(* Logix 5000 project; controller Safety vendor 1 type 14 code 86 rev 19.11; software revision 19.01; part 8 of 17 *)
(* tags used below, declared in another part *)
   ESTOP_x201PB040 : DCI_STOP;   // OS1 Line EStop Pushbutton
   ESTOP_x201PB040_Flt : ALIAS FOR Flt_Estops.0;   // OS1 Line EStop Pushbutton Fault ( 1= Fault)
   ESTOP_x211PB040 : DCI_STOP;   // OS2 Line EStop Pushbutton
   ESTOP_x211PB040_Flt : ALIAS FOR Flt_Estops.1;   // OS2 Line EStop Pushbutton Fault ( 1= Fault)
   ESTOP_x221PB040 : DCI_STOP;   // OS3 Line EStop Pushbutton
   ESTOP_x221PB040_Flt : ALIAS FOR Flt_Estops.2;   // OS3 Line EStop Pushbutton Fault ( 1= Fault)
   ESTOP_x231PB040 : DCI_STOP;   // OS4N Line EStop Pushbutton
   ESTOP_x231PB040_Flt : ALIAS FOR Flt_Estops.3;   // OS4N Line EStop Pushbutton Fault ( 1= Fault)
   ESTOP_x241PB040 : DCI_STOP;   // OS4S Line EStop Pushbutton
   ESTOP_x241PB040_Flt : ALIAS FOR Flt_Estops.4;   // OS4S Line EStop Pushbutton Fault ( 1= Fault)
   ESTOP_x251PB040 : DCI_STOP;   // OS5 Line EStop Pushbutton
   ESTOP_x251PB040_Flt : ALIAS FOR Flt_Estops.5;   // OS5 Line EStop Pushbutton Fault ( 1= Fault)
   ESTOP_x261PB040 : DCI_STOP;   // OS6 Line EStop Pushbutton
   ESTOP_x261PB040_Flt : ALIAS FOR Flt_Estops.6;   // OS6 Line EStop Pushbutton Fault ( 1= Fault)
   ESTOP_x271PB040 : DCI_STOP;   // OS8 Line EStop Pushbutton
   ESTOP_x271PB040_Flt : ALIAS FOR Flt_Estops.7;   // OS8 Line EStop Pushbutton Fault ( 1= Fault)
   ESTOP_x281PB040 : DCI_STOP;   // OS9 Line EStop Pushbutton
   ESTOP_x301PB040 : DCI_STOP;   // OS13 Line EStop Pushbutton
   ESTOP_x311PB040 : DCI_STOP;   // OS14 Line EStop Pushbutton
   ESTOP_x311PB130 : DCI_STOP;   // OS14 Shear Estop Pushbutton
   ESTOP_x321PB040 : DCI_STOP;   // OS15 Line EStop Pushbutton
   ESTOP_x331PB040 : DCI_STOP;   // OS16 Line EStop Pushbutton
   ESTOP_x480PB550 : DCI_STOP;   // DPD (In Pit) Line EStop Pushbutton
   ESTOP_x519LS470 : DCI_STOP;   // G1 Tripwire Line EStop
   ESTOP_x533PB470 : DCI_STOP;   // H1 Line EStop Pushbutton
   Line_TotalMode : BOOL;   // Line TOTAL Mode ( 1= Total Mode) (0 = Coil to Coil)
   LineSts : UDT_SysStatus;
   OS1_EstopRstCmd : BOOL;   // OS1 Estop Reset Command ( 1= Reset Cmd)
   OS1_FltRstCmd : BOOL;   // OS1 Fault Reset Command ( 1= Reset Cmd)
   OS1_No_EStops : BOOL;   // OS1 No Estops ( 1= OK)
   OS2_EstopRstCmd : BOOL;   // OS2 Estop Reset Command ( 1= Reset Cmd)
   OS2_FltRstCmd : BOOL;   // OS2 Fault Reset Command ( 1= Reset Cmd)
   OS2_No_EStops : BOOL;   // OS2 No Estops ( 1= OK)
   OS3_EstopRstCmd : BOOL;   // OS3 Estop Reset Command ( 1= Reset Cmd)
   OS3_FltRstCmd : BOOL;   // OS3 Fault Reset Command ( 1= Reset Cmd)
   OS3_No_EStops : BOOL;   // OS3 No Estops ( 1= OK)
   OS4_EstopRstCmd : BOOL;   // OS4 Estop Reset Command ( 1= Reset Cmd)
   OS4_FltRstCmd : BOOL;   // OS4 Fault Reset Command ( 1= Reset Cmd)
   OS4_No_EStops : BOOL;   // OS4 No Estops ( 1= OK)
   OS5_EstopRstCmd : BOOL;   // OS5 Estop Reset Command ( 1= Reset Cmd)
   OS5_FltRstCmd : BOOL;   // OS5 Fault Reset Command ( 1= Reset Cmd)
   OS5_No_EStops : BOOL;   // OS5 No Estops ( 1= OK)
   OS6_EstopRstCmd : BOOL;   // OS6 Estop Reset Command ( 1= Reset Cmd)
   OS6_FltRstCmd : BOOL;   // OS6 Fault Reset Command ( 1= Reset Cmd)
   OS6_No_EStops : BOOL;   // OS6 No Estops ( 1= OK)
   OS8_EstopRstCmd : BOOL;   // OS8 Estop Reset Command ( 1= Reset Cmd)
   OS8_FltRstCmd : BOOL;   // OS8 Fault Reset Command ( 1= Reset Cmd)
   OS8_No_EStops : BOOL;   // OS8 No Estops ( 1= OK)
   x201PB040a : ALIAS FOR OS1:1:I.Pt00Data;   // Line Emergency Stop PB
   x201PB040b : ALIAS FOR OS1:1:I.Pt01Data;   // Line Emergency Stop PB
   x211PB040a : ALIAS FOR OS2:1:I.Pt00Data;   // Line Emergency Stop PB
   x211PB040b : ALIAS FOR OS2:1:I.Pt01Data;   // Line Emergency Stop PB
   x221PB040a : ALIAS FOR OS3:1:I.Pt00Data;   // Emergency Stop PB
   x221PB040b : ALIAS FOR OS3:1:I.Pt01Data;   // Emergency Stop PB
   x231PB040a : ALIAS FOR OS4N:1:I.Pt00Data;   // Emergency Stop PB
   x231PB040b : ALIAS FOR OS4N:1:I.Pt01Data;   // Emergency Stop PB
   x241PB040a : ALIAS FOR OS4S:1:I.Pt00Data;   // Emergency Stop PBMc_A_Run1_A
   x241PB040b : ALIAS FOR OS4S:1:I.Pt01Data;   // Emergency Stop PBMc_A_Run1_A
   x251PB040a : ALIAS FOR OS5:1:I.Pt00Data;   // Emergency Stop PB
   x251PB040b : ALIAS FOR OS5:1:I.Pt01Data;   // Emergency Stop PB
   x261PB040a : ALIAS FOR OS6:1:I.Pt00Data;   // Emergency Stop PB
   x261PB040b : ALIAS FOR OS6:1:I.Pt01Data;   // Emergency Stop PB
   x271PB040a : ALIAS FOR OS8:1:I.Pt00Data;   // Emergency Stop PB
   x271PB040b : ALIAS FOR OS8:1:I.Pt01Data;   // Emergency Stop PB

PROGRAM Estops   (* main routine A00_Main *)
// Estop PB's

ROUTINE A00_Main   (* ladder *)
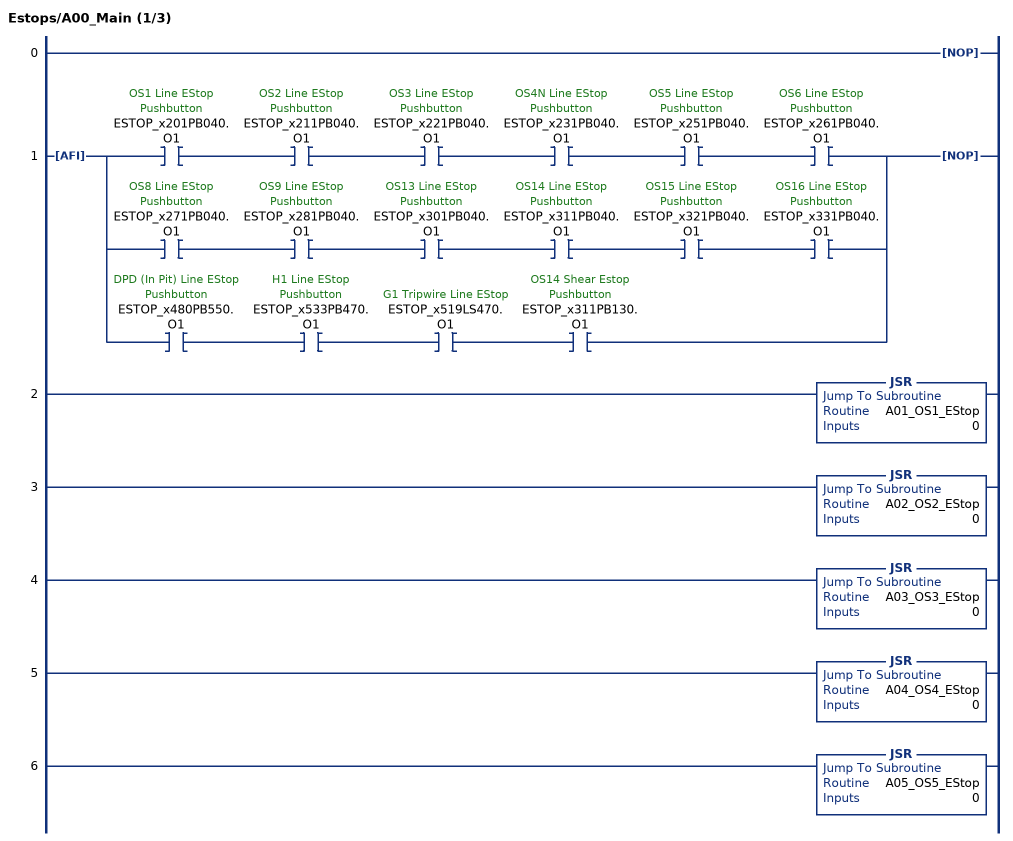
   0: NOP();
   1: AFI()[XIC(ESTOP_x201PB040.O1) XIC(ESTOP_x211PB040.O1) XIC(ESTOP_x221PB040.O1) XIC(ESTOP_x231PB040.O1) XIC(ESTOP_x251PB040.O1) XIC(ESTOP_x261PB040.O1) ,XIC(ESTOP_x271PB040.O1) XIC(ESTOP_x281PB040.O1) XIC(ESTOP_x301PB040.O1) XIC(ESTOP_x311PB040.O1) XIC(ESTOP_x321PB040.O1) XIC(ESTOP_x331PB040.O1) ,XIC(ESTOP_x480PB550.O1) XIC(ESTOP_x533PB470.O1) XIC(ESTOP_x519LS470.O1) XIC(ESTOP_x311PB130.O1) ]NOP();
   2: JSR(A01_OS1_EStop,0);
   3: JSR(A02_OS2_EStop,0);
   4: JSR(A03_OS3_EStop,0);
   5: JSR(A04_OS4_EStop,0);
   6: JSR(A05_OS5_EStop,0);
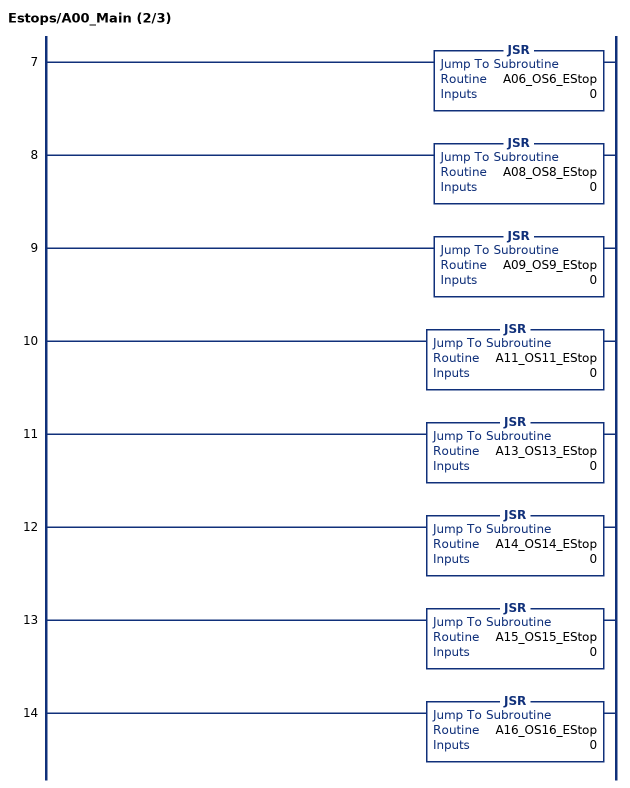
   7: JSR(A06_OS6_EStop,0);
   8: JSR(A08_OS8_EStop,0);
   9: JSR(A09_OS9_EStop,0);
   10: JSR(A11_OS11_EStop,0);
   11: JSR(A13_OS13_EStop,0);
   12: JSR(A14_OS14_EStop,0);
   13: JSR(A15_OS15_EStop,0);
   14: JSR(A16_OS16_EStop,0);
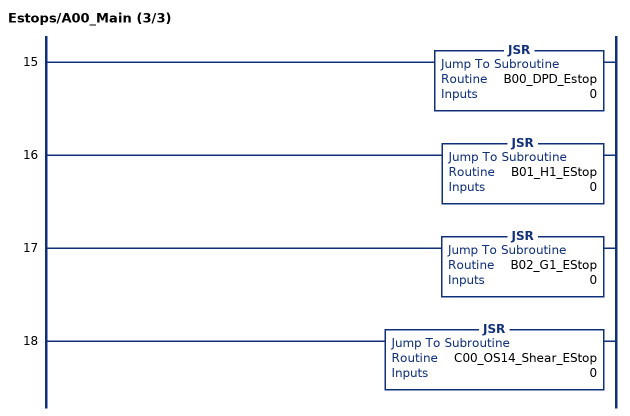
   15: JSR(B00_DPD_Estop,0);
   16: JSR(B01_H1_EStop,0);
   17: JSR(B02_G1_EStop,0);
   18: JSR(C00_OS14_Shear_EStop,0);
END_ROUTINE

ROUTINE A01_OS1_EStop   (* ladder *)
// OS1 Estops
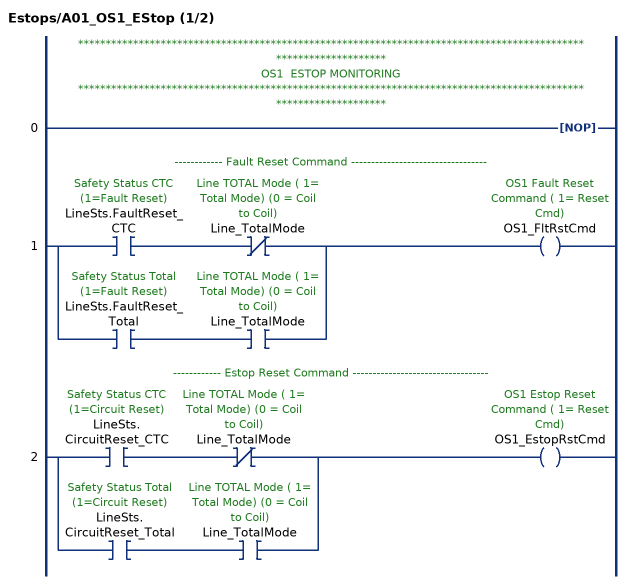
   // ****************************************************************************************************************
   // OS1  ESTOP MONITORING
   // ****************************************************************************************************************
   0: NOP();
   // ------------ Fault Reset Command ----------------------------------
   1: [XIC(LineSts.FaultReset_CTC) XIO(Line_TotalMode) ,XIC(LineSts.FaultReset_Total) XIC(Line_TotalMode) ]OTE(OS1_FltRstCmd);
   // ------------ Estop Reset Command ----------------------------------
   2: [XIC(LineSts.CircuitReset_CTC) XIO(Line_TotalMode) ,XIC(LineSts.CircuitReset_Total) XIC(Line_TotalMode) ]OTE(OS1_EstopRstCmd);
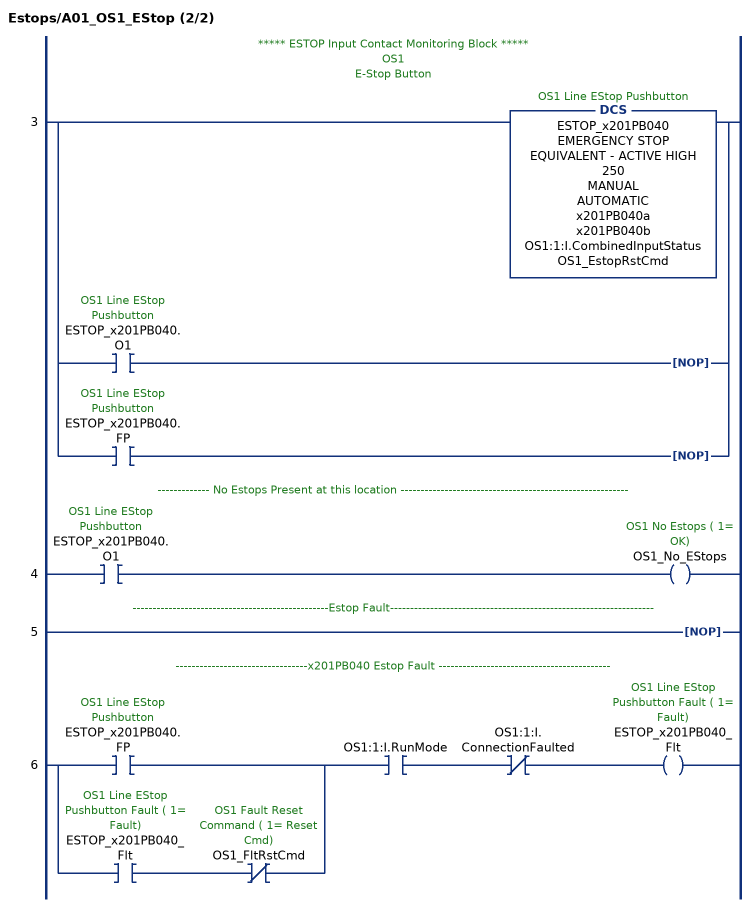
   // ***** ESTOP Input Contact Monitoring Block *****
   // OS1
   // E-Stop Button
   3: [DCS(ESTOP_x201PB040,EMERGENCY STOP,EQUIVALENT - ACTIVE HIGH,250,MANUAL,AUTOMATIC,x201PB040a,x201PB040b,OS1:1:I.CombinedInputStatus,OS1_EstopRstCmd) ,XIC(ESTOP_x201PB040.O1) NOP() ,XIC(ESTOP_x201PB040.FP) NOP() ];
   // ------------- No Estops Present at this location ---------------------------------------------------------
   4: XIC(ESTOP_x201PB040.O1)OTE(OS1_No_EStops);
   // -------------------------------------------------Estop Fault------------------------------------------------------------------
   5: NOP();
   // ---------------------------------x201PB040 Estop Fault -------------------------------------------
   6: [XIC(ESTOP_x201PB040.FP) ,XIC(ESTOP_x201PB040_Flt) XIO(OS1_FltRstCmd) ]XIC(OS1:1:I.RunMode)XIO(OS1:1:I.ConnectionFaulted)OTE(ESTOP_x201PB040_Flt);
END_ROUTINE

ROUTINE A02_OS2_EStop   (* ladder *)
// OS2 Estops
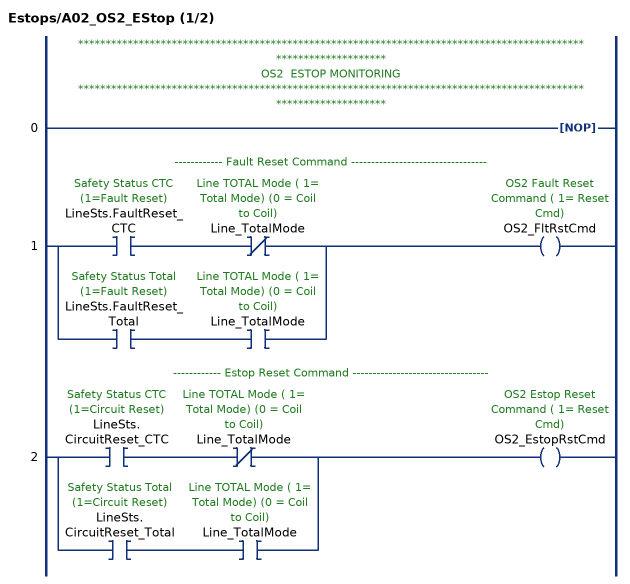
   // ****************************************************************************************************************
   // OS2  ESTOP MONITORING
   // ****************************************************************************************************************
   0: NOP();
   // ------------ Fault Reset Command ----------------------------------
   1: [XIC(LineSts.FaultReset_CTC) XIO(Line_TotalMode) ,XIC(LineSts.FaultReset_Total) XIC(Line_TotalMode) ]OTE(OS2_FltRstCmd);
   // ------------ Estop Reset Command ----------------------------------
   2: [XIC(LineSts.CircuitReset_CTC) XIO(Line_TotalMode) ,XIC(LineSts.CircuitReset_Total) XIC(Line_TotalMode) ]OTE(OS2_EstopRstCmd);
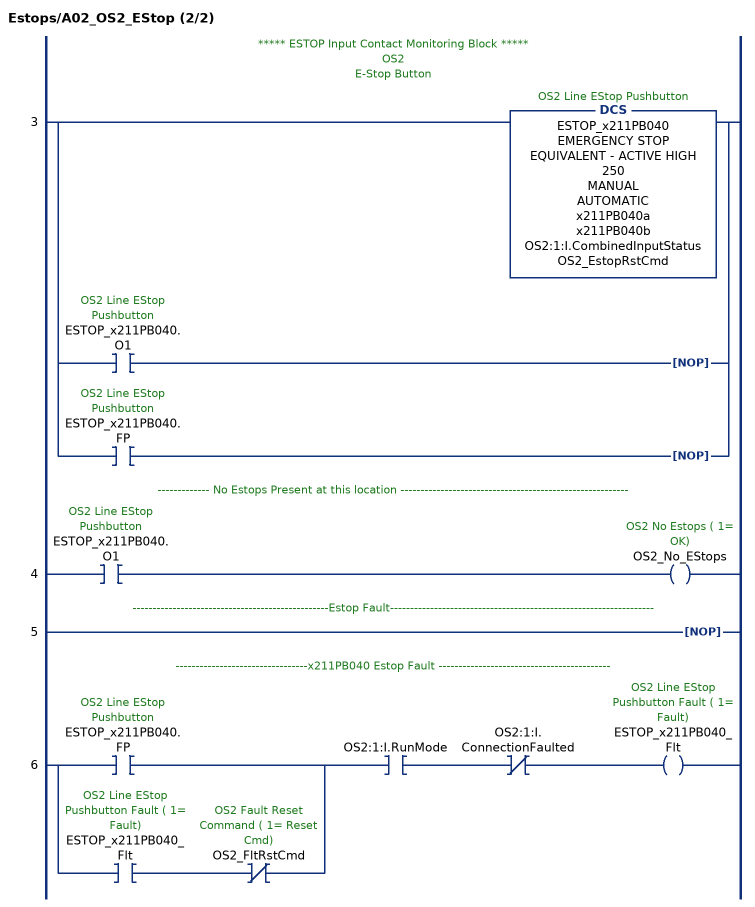
   // ***** ESTOP Input Contact Monitoring Block *****
   // OS2
   // E-Stop Button
   3: [DCS(ESTOP_x211PB040,EMERGENCY STOP,EQUIVALENT - ACTIVE HIGH,250,MANUAL,AUTOMATIC,x211PB040a,x211PB040b,OS2:1:I.CombinedInputStatus,OS2_EstopRstCmd) ,XIC(ESTOP_x211PB040.O1) NOP() ,XIC(ESTOP_x211PB040.FP) NOP() ];
   // ------------- No Estops Present at this location ---------------------------------------------------------
   4: XIC(ESTOP_x211PB040.O1)OTE(OS2_No_EStops);
   // -------------------------------------------------Estop Fault------------------------------------------------------------------
   5: NOP();
   // ---------------------------------x211PB040 Estop Fault -------------------------------------------
   6: [XIC(ESTOP_x211PB040.FP) ,XIC(ESTOP_x211PB040_Flt) XIO(OS2_FltRstCmd) ]XIC(OS2:1:I.RunMode)XIO(OS2:1:I.ConnectionFaulted)OTE(ESTOP_x211PB040_Flt);
END_ROUTINE

ROUTINE A03_OS3_EStop   (* ladder *)
// OS3 Estops
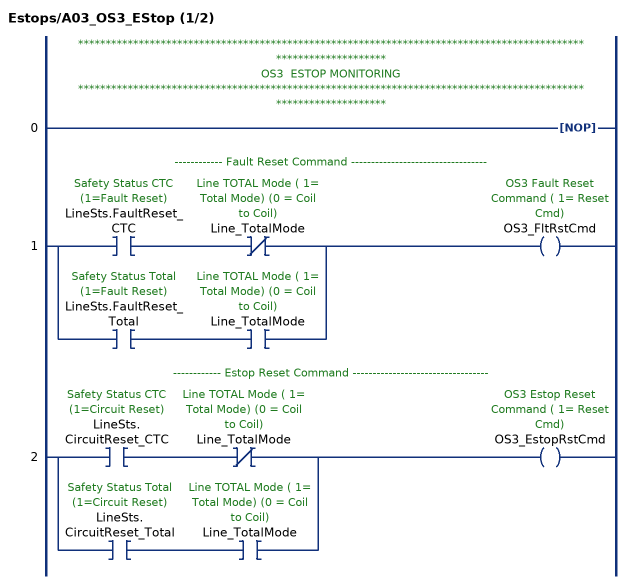
   // ****************************************************************************************************************
   // OS3  ESTOP MONITORING
   // ****************************************************************************************************************
   0: NOP();
   // ------------ Fault Reset Command ----------------------------------
   1: [XIC(LineSts.FaultReset_CTC) XIO(Line_TotalMode) ,XIC(LineSts.FaultReset_Total) XIC(Line_TotalMode) ]OTE(OS3_FltRstCmd);
   // ------------ Estop Reset Command ----------------------------------
   2: [XIC(LineSts.CircuitReset_CTC) XIO(Line_TotalMode) ,XIC(LineSts.CircuitReset_Total) XIC(Line_TotalMode) ]OTE(OS3_EstopRstCmd);
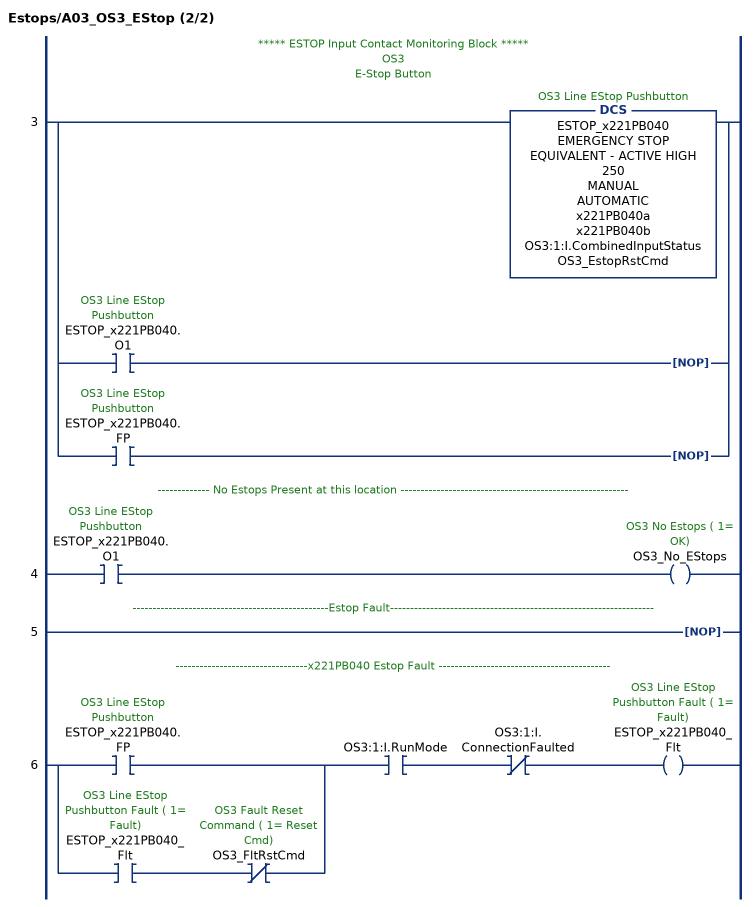
   // ***** ESTOP Input Contact Monitoring Block *****
   // OS3
   // E-Stop Button
   3: [DCS(ESTOP_x221PB040,EMERGENCY STOP,EQUIVALENT - ACTIVE HIGH,250,MANUAL,AUTOMATIC,x221PB040a,x221PB040b,OS3:1:I.CombinedInputStatus,OS3_EstopRstCmd) ,XIC(ESTOP_x221PB040.O1) NOP() ,XIC(ESTOP_x221PB040.FP) NOP() ];
   // ------------- No Estops Present at this location ---------------------------------------------------------
   4: XIC(ESTOP_x221PB040.O1)OTE(OS3_No_EStops);
   // -------------------------------------------------Estop Fault------------------------------------------------------------------
   5: NOP();
   // ---------------------------------x221PB040 Estop Fault -------------------------------------------
   6: [XIC(ESTOP_x221PB040.FP) ,XIC(ESTOP_x221PB040_Flt) XIO(OS3_FltRstCmd) ]XIC(OS3:1:I.RunMode)XIO(OS3:1:I.ConnectionFaulted)OTE(ESTOP_x221PB040_Flt);
END_ROUTINE

ROUTINE A04_OS4_EStop   (* ladder *)
// OS4N/S Estops
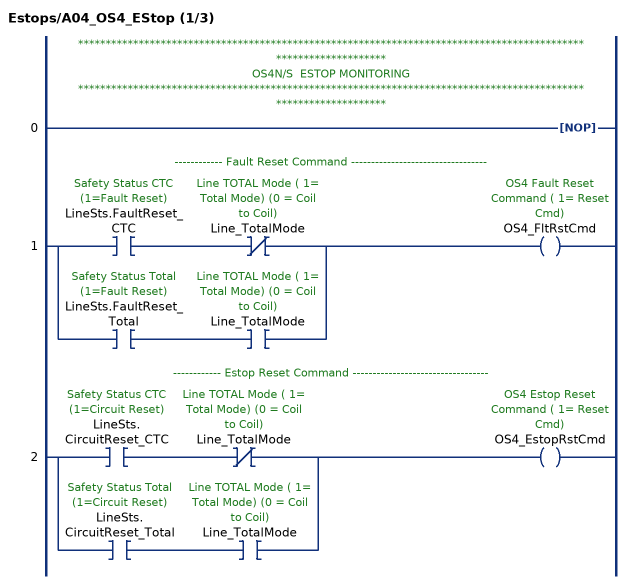
   // ****************************************************************************************************************
   // OS4N/S  ESTOP MONITORING
   // ****************************************************************************************************************
   0: NOP();
   // ------------ Fault Reset Command ----------------------------------
   1: [XIC(LineSts.FaultReset_CTC) XIO(Line_TotalMode) ,XIC(LineSts.FaultReset_Total) XIC(Line_TotalMode) ]OTE(OS4_FltRstCmd);
   // ------------ Estop Reset Command ----------------------------------
   2: [XIC(LineSts.CircuitReset_CTC) XIO(Line_TotalMode) ,XIC(LineSts.CircuitReset_Total) XIC(Line_TotalMode) ]OTE(OS4_EstopRstCmd);
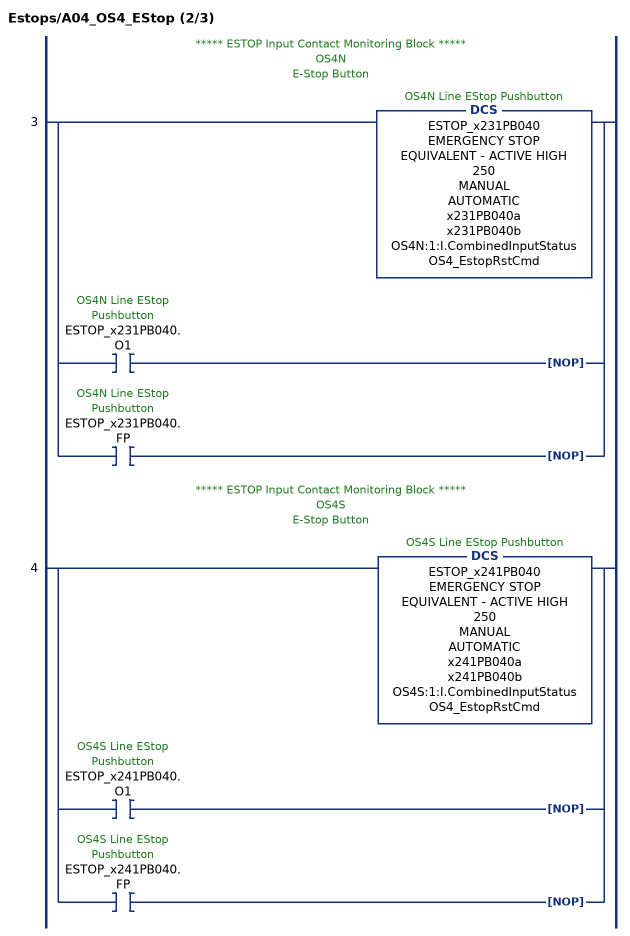
   // ***** ESTOP Input Contact Monitoring Block *****
   // OS4N
   // E-Stop Button
   3: [DCS(ESTOP_x231PB040,EMERGENCY STOP,EQUIVALENT - ACTIVE HIGH,250,MANUAL,AUTOMATIC,x231PB040a,x231PB040b,OS4N:1:I.CombinedInputStatus,OS4_EstopRstCmd) ,XIC(ESTOP_x231PB040.O1) NOP() ,XIC(ESTOP_x231PB040.FP) NOP() ];
   // ***** ESTOP Input Contact Monitoring Block *****
   // OS4S
   // E-Stop Button
   4: [DCS(ESTOP_x241PB040,EMERGENCY STOP,EQUIVALENT - ACTIVE HIGH,250,MANUAL,AUTOMATIC,x241PB040a,x241PB040b,OS4S:1:I.CombinedInputStatus,OS4_EstopRstCmd) ,XIC(ESTOP_x241PB040.O1) NOP() ,XIC(ESTOP_x241PB040.FP) NOP() ];
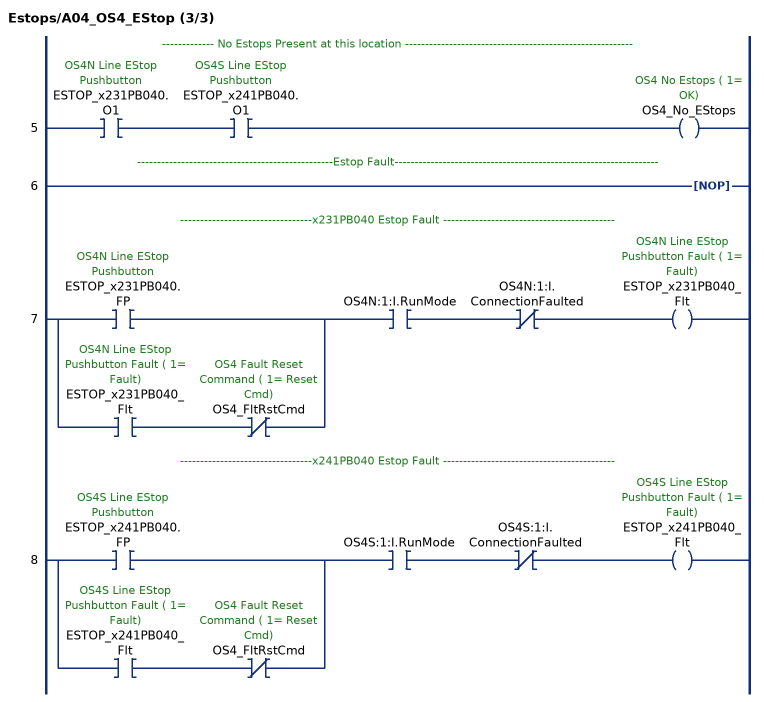
   // ------------- No Estops Present at this location ---------------------------------------------------------
   5: XIC(ESTOP_x231PB040.O1)XIC(ESTOP_x241PB040.O1)OTE(OS4_No_EStops);
   // -------------------------------------------------Estop Fault------------------------------------------------------------------
   6: NOP();
   // ---------------------------------x231PB040 Estop Fault -------------------------------------------
   7: [XIC(ESTOP_x231PB040.FP) ,XIC(ESTOP_x231PB040_Flt) XIO(OS4_FltRstCmd) ]XIC(OS4N:1:I.RunMode)XIO(OS4N:1:I.ConnectionFaulted)OTE(ESTOP_x231PB040_Flt);
   // ---------------------------------x241PB040 Estop Fault -------------------------------------------
   8: [XIC(ESTOP_x241PB040.FP) ,XIC(ESTOP_x241PB040_Flt) XIO(OS4_FltRstCmd) ]XIC(OS4S:1:I.RunMode)XIO(OS4S:1:I.ConnectionFaulted)OTE(ESTOP_x241PB040_Flt);
END_ROUTINE

ROUTINE A05_OS5_EStop   (* ladder *)
// OS5 Estops
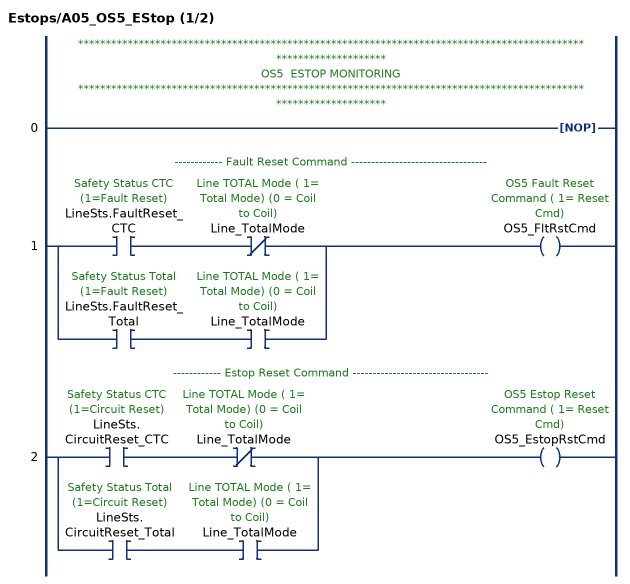
   // ****************************************************************************************************************
   // OS5  ESTOP MONITORING
   // ****************************************************************************************************************
   0: NOP();
   // ------------ Fault Reset Command ----------------------------------
   1: [XIC(LineSts.FaultReset_CTC) XIO(Line_TotalMode) ,XIC(LineSts.FaultReset_Total) XIC(Line_TotalMode) ]OTE(OS5_FltRstCmd);
   // ------------ Estop Reset Command ----------------------------------
   2: [XIC(LineSts.CircuitReset_CTC) XIO(Line_TotalMode) ,XIC(LineSts.CircuitReset_Total) XIC(Line_TotalMode) ]OTE(OS5_EstopRstCmd);
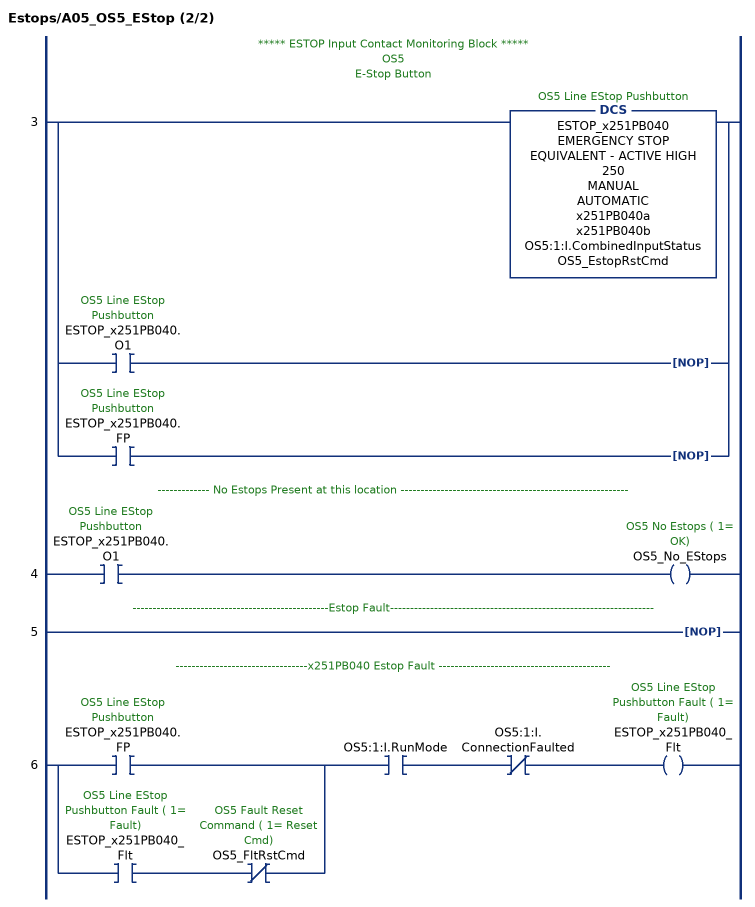
   // ***** ESTOP Input Contact Monitoring Block *****
   // OS5
   // E-Stop Button
   3: [DCS(ESTOP_x251PB040,EMERGENCY STOP,EQUIVALENT - ACTIVE HIGH,250,MANUAL,AUTOMATIC,x251PB040a,x251PB040b,OS5:1:I.CombinedInputStatus,OS5_EstopRstCmd) ,XIC(ESTOP_x251PB040.O1) NOP() ,XIC(ESTOP_x251PB040.FP) NOP() ];
   // ------------- No Estops Present at this location ---------------------------------------------------------
   4: XIC(ESTOP_x251PB040.O1)OTE(OS5_No_EStops);
   // -------------------------------------------------Estop Fault------------------------------------------------------------------
   5: NOP();
   // ---------------------------------x251PB040 Estop Fault -------------------------------------------
   6: [XIC(ESTOP_x251PB040.FP) ,XIC(ESTOP_x251PB040_Flt) XIO(OS5_FltRstCmd) ]XIC(OS5:1:I.RunMode)XIO(OS5:1:I.ConnectionFaulted)OTE(ESTOP_x251PB040_Flt);
END_ROUTINE

ROUTINE A06_OS6_EStop   (* ladder *)
// OS6 Estops
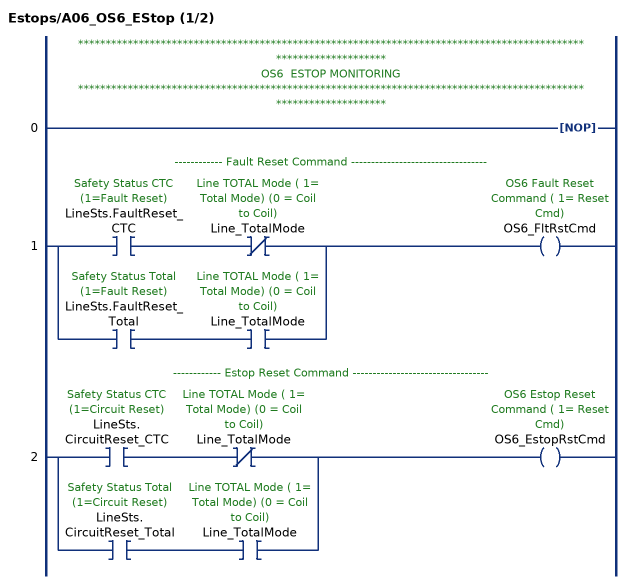
   // ****************************************************************************************************************
   // OS6  ESTOP MONITORING
   // ****************************************************************************************************************
   0: NOP();
   // ------------ Fault Reset Command ----------------------------------
   1: [XIC(LineSts.FaultReset_CTC) XIO(Line_TotalMode) ,XIC(LineSts.FaultReset_Total) XIC(Line_TotalMode) ]OTE(OS6_FltRstCmd);
   // ------------ Estop Reset Command ----------------------------------
   2: [XIC(LineSts.CircuitReset_CTC) XIO(Line_TotalMode) ,XIC(LineSts.CircuitReset_Total) XIC(Line_TotalMode) ]OTE(OS6_EstopRstCmd);
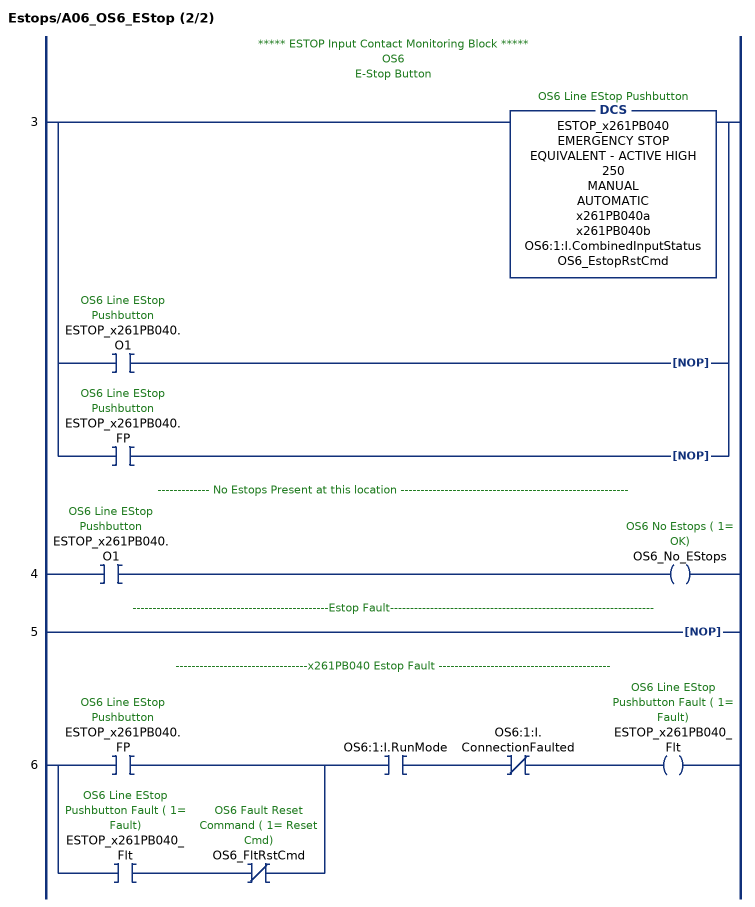
   // ***** ESTOP Input Contact Monitoring Block *****
   // OS6
   // E-Stop Button
   3: [DCS(ESTOP_x261PB040,EMERGENCY STOP,EQUIVALENT - ACTIVE HIGH,250,MANUAL,AUTOMATIC,x261PB040a,x261PB040b,OS6:1:I.CombinedInputStatus,OS6_EstopRstCmd) ,XIC(ESTOP_x261PB040.O1) NOP() ,XIC(ESTOP_x261PB040.FP) NOP() ];
   // ------------- No Estops Present at this location ---------------------------------------------------------
   4: XIC(ESTOP_x261PB040.O1)OTE(OS6_No_EStops);
   // -------------------------------------------------Estop Fault------------------------------------------------------------------
   5: NOP();
   // ---------------------------------x261PB040 Estop Fault -------------------------------------------
   6: [XIC(ESTOP_x261PB040.FP) ,XIC(ESTOP_x261PB040_Flt) XIO(OS6_FltRstCmd) ]XIC(OS6:1:I.RunMode)XIO(OS6:1:I.ConnectionFaulted)OTE(ESTOP_x261PB040_Flt);
END_ROUTINE

ROUTINE A08_OS8_EStop   (* ladder *)
// OS8 Estops
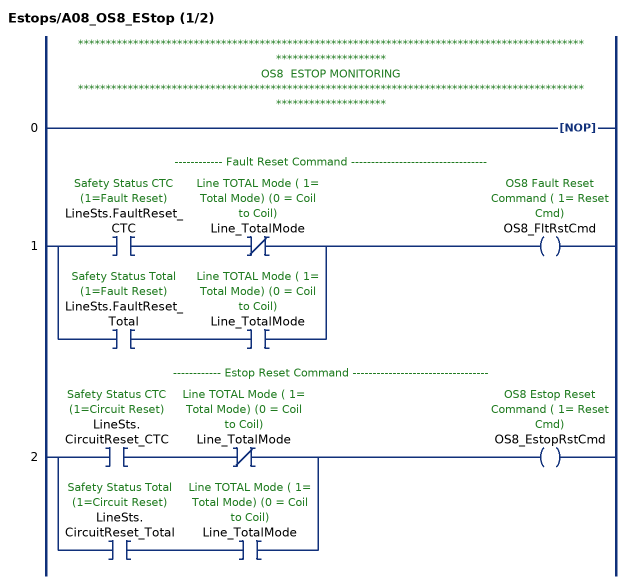
   // ****************************************************************************************************************
   // OS8  ESTOP MONITORING
   // ****************************************************************************************************************
   0: NOP();
   // ------------ Fault Reset Command ----------------------------------
   1: [XIC(LineSts.FaultReset_CTC) XIO(Line_TotalMode) ,XIC(LineSts.FaultReset_Total) XIC(Line_TotalMode) ]OTE(OS8_FltRstCmd);
   // ------------ Estop Reset Command ----------------------------------
   2: [XIC(LineSts.CircuitReset_CTC) XIO(Line_TotalMode) ,XIC(LineSts.CircuitReset_Total) XIC(Line_TotalMode) ]OTE(OS8_EstopRstCmd);
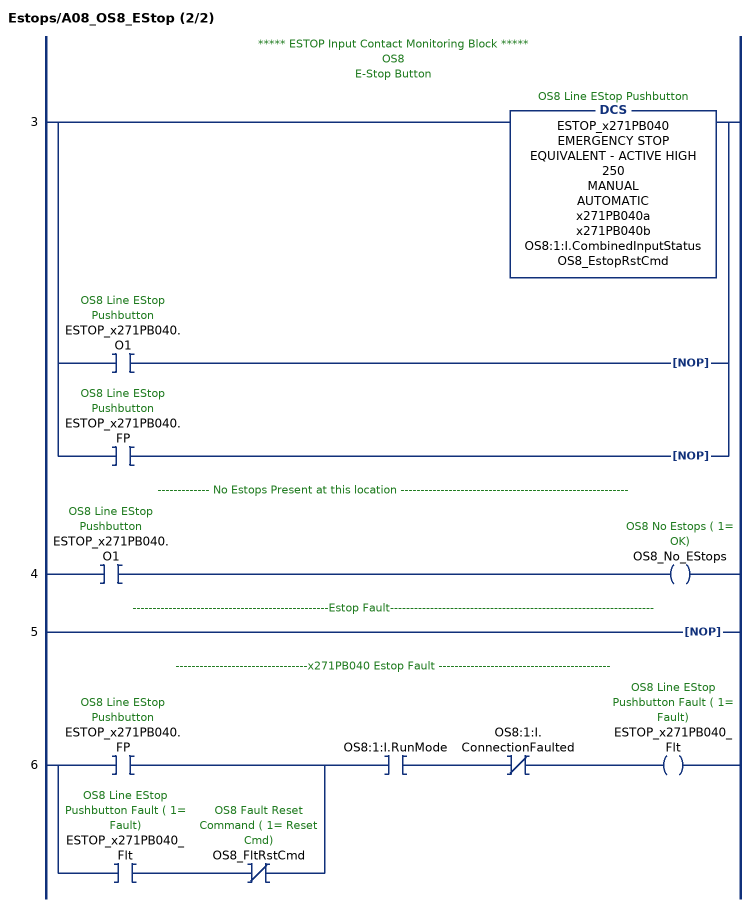
   // ***** ESTOP Input Contact Monitoring Block *****
   // OS8
   // E-Stop Button
   3: [DCS(ESTOP_x271PB040,EMERGENCY STOP,EQUIVALENT - ACTIVE HIGH,250,MANUAL,AUTOMATIC,x271PB040a,x271PB040b,OS8:1:I.CombinedInputStatus,OS8_EstopRstCmd) ,XIC(ESTOP_x271PB040.O1) NOP() ,XIC(ESTOP_x271PB040.FP) NOP() ];
   // ------------- No Estops Present at this location ---------------------------------------------------------
   4: XIC(ESTOP_x271PB040.O1)OTE(OS8_No_EStops);
   // -------------------------------------------------Estop Fault------------------------------------------------------------------
   5: NOP();
   // ---------------------------------x271PB040 Estop Fault -------------------------------------------
   6: [XIC(ESTOP_x271PB040.FP) ,XIC(ESTOP_x271PB040_Flt) XIO(OS8_FltRstCmd) ]XIC(OS8:1:I.RunMode)XIO(OS8:1:I.ConnectionFaulted)OTE(ESTOP_x271PB040_Flt);
END_ROUTINE
